(* IEC 61131-3 sources: SRCI/RobotLibrary/Library/POUs/Additional/MC_OpenBrake, 1 file *)

(* ---- MC_OpenBrakeFB.st ---- *)
/// Release robot arm’s brakes.
FUNCTION_BLOCK MC_OpenBrakeFB EXTENDS RobotLibraryBaseExecuteFB
// -------------------------------------------------------------------------
//  SRCI Robot Library
// -------------------------------------------------------------------------
//
//  Object:      OpenBrakeFB
//  Author:      Thorsten Brach
//  Date:        2024-06-01
//
//  Description:
//
//
//  Copyright:
//    (C) 2024 Thorsten Brach. All rights reserved
//             Licensed under the LGPL-3.0 license.
//
//  Disclaimer:
//    This project is provided without any guarantee and can be used for
//    private and commercial purposes. Any use is at the user’s
//    own risk and responsibility.
//
// -------------------------------------------------------------------------
VAR_INPUT
  /// Command parameter
  ParCmd             : OpenBrakeParCmd;
END_VAR

VAR_OUTPUT
  /// Command is transferred and confirmed by the RC
  CommandBuffered   : BOOL;
  /// Receiving of input parameter values has been acknowledged by RC
  ParameterAccepted : BOOL;
  /// Command output
  OutCmd            : OpenBrakeOutCmd;
END_VAR

VAR
  /// internal copy of command parameter
 _parCmd             : OpenBrakeParCmd;
  /// command data to send
 _command            : OpenBrakeSendData;
  /// response data received
 _response           : OpenBrakeRecvData;
END_VAR

  SUPER^(AxesGroup := AxesGroup);

END_FUNCTION_BLOCK

METHOD INTERNAL CheckAddParameter : BOOL
VAR_INPUT
  /// Payload pointer
  PayloadPtr : UDINT;
END_VAR
VAR
  /// Payload as byte array
  Payload    : ARRAY [1..SIZEOF(_command)] OF BYTE;
  /// Null Byte array
  Null       : ARRAY [1..SIZEOF(_command)] OF BYTE;
  /// Data length to compare
  DataLen    : UDINT;
END_VAR

  // Payload pointer must be decreased by one byte, because ADR(Payload) is already one byte !
  PayloadPtr := LIMIT (0, PayloadPtr - 1, SIZEOF(Payload) -1);
  // Convert command struct to payload array
  SysDepMemCpy( pDest := ADR(Payload), pSrc := ADR(_command), DataLen := SIZEOF(_command));
  // Calculate the data length to compare - at least one byte must be compared !
  DataLen := LIMIT(1, SIZEOF(Payload) - PayloadPtr, SIZEOF(Payload));
  // Compare Payload-Array with Null-Byte-Array
  CheckAddParameter := SysDepMemCmp( pData1 := ADR(Payload) + PayloadPtr , pData2 := ADR(Null), DataLen := DataLen) <>  RobotLibraryConstants.OK ;

END_METHOD

METHOD PROTECTED CheckFunctionSupported : BOOL
VAR_IN_OUT
  /// Robot assignment of function
  AxesGroup : AxesGroup;
END_VAR

  CheckFunctionSupported := AxesGroup.State.RobotData.RCSupportedFunctions.OpenBrake;

  IF ( NOT CheckFunctionSupported )
  THEN
    // call base implementation for set error and create log entry
    SUPER^.CheckFunctionSupported(AxesGroup := AxesGroup);
  END_IF

END_METHOD

METHOD PROTECTED CheckParameterChanged : BOOL
VAR_IN_OUT
  /// Robot assignment of function
  AxesGroup    : AxesGroup;
END_VAR

  // Check ParCmd Size is > 0, because MemCmp does not work correctly with size = 0
  IF (SIZEOF(ParCmd) = 0) OR (_stepCmd = 0)
  THEN
    RETURN;
  END_IF

  // compare memory
  _parameterChanged := ( SysDepMemCmp(pData1 := ADR(ParCmd), pData2 := ADR(_parCmd), DataLen := SIZEOF(ParCmd)) <> RobotLibraryConstants.OK );

  // check parameter valid ?
  _parameterValid   := CheckParameterValid( AxesGroup := AxesGroup );

  IF ((  _parameterChanged        )  AND
      (  _parameterValid          )) OR
      (  _parameterUpdateInternal )
  THEN
    // reset internal flag for send parameter update
   _parameterUpdateInternal := FALSE;
    // update internal copy of parameters
   _parCmd := ParCmd;
    // inc parameter sequence
   _command.ParSeq := _command.ParSeq + 1;
    // update command data
    CommandData := CreateCommandPayload(AxesGroup := AxesGroup); // ( Access via reference to rCommandFB in ACR )
    // notify active command register
    AxesGroup.Acyclic.ActiveCommandRegister.NotifyParameterChanged := _uniqueID;
    // Reset parameter accepted flag
    ParameterAccepted := FALSE;
  END_IF

END_METHOD

METHOD PROTECTED CheckParameterValid : BOOL
VAR_IN_OUT
  /// Robot assignment of function
  AxesGroup : AxesGroup;
END_VAR

  CheckParameterValid := TRUE;

  // Check ParCmd.ParCmd.RobotAxesBrakeRelease.AxisJ1 valid ?
  IF (( ParCmd.RobotAxesBrakeRelease.AxisJ1) AND ( NOT AxesGroup.State.RobotData.AxisJointUsed.J1 ))
  THEN
    // Parameter not valid
    CheckParameterValid := FALSE;
    // Set error
    ErrorID := RobotLibraryErrorIdEnum.ERR_INVALID_PAR_CMD;
    // Create log entry
    CreateLogMessagePara1 ( Timestamp   := AxesGroup.State.SystemTime,
                            MessageType := MessageType.CMD,
                            Severity    := Severity.ERROR,
                            MessageCode := ErrorID,
                            MessageText := 'Invalid Parameter ParCmd.RobotAxesBrakeRelease.AxisJ1 = {1}',
                            Para1       :=  BOOL_TO_STRING(ParCmd.RobotAxesBrakeRelease.AxisJ1));
    RETURN;
  END_IF

  // Check ParCmd.ParCmd.RobotAxesBrakeRelease.AxisJ2 valid ?
  IF (( ParCmd.RobotAxesBrakeRelease.AxisJ2) AND ( NOT AxesGroup.State.RobotData.AxisJointUsed.J2 ))
  THEN
    // Parameter not valid
    CheckParameterValid := FALSE;
    // Set error
    ErrorID := RobotLibraryErrorIdEnum.ERR_INVALID_PAR_CMD;
    // Create log entry
    CreateLogMessagePara1 ( Timestamp   := AxesGroup.State.SystemTime,
                            MessageType := MessageType.CMD,
                            Severity    := Severity.ERROR,
                            MessageCode := ErrorID,
                            MessageText := 'Invalid Parameter ParCmd.RobotAxesBrakeRelease.AxisJ2 = {1}',
                            Para1       :=  BOOL_TO_STRING(ParCmd.RobotAxesBrakeRelease.AxisJ2));
    RETURN;
  END_IF

  // Check ParCmd.ParCmd.RobotAxesBrakeRelease.AxisJ3 valid ?
  IF (( ParCmd.RobotAxesBrakeRelease.AxisJ3) AND ( NOT AxesGroup.State.RobotData.AxisJointUsed.J3 ))
  THEN
    // Parameter not valid
    CheckParameterValid := FALSE;
    // Set error
    ErrorID := RobotLibraryErrorIdEnum.ERR_INVALID_PAR_CMD;
    // Create log entry
    CreateLogMessagePara1 ( Timestamp   := AxesGroup.State.SystemTime,
                            MessageType := MessageType.CMD,
                            Severity    := Severity.ERROR,
                            MessageCode := ErrorID,
                            MessageText := 'Invalid Parameter ParCmd.RobotAxesBrakeRelease.AxisJ3 = {1}',
                            Para1       :=  BOOL_TO_STRING(ParCmd.RobotAxesBrakeRelease.AxisJ3));
    RETURN;
  END_IF

  // Check ParCmd.ParCmd.RobotAxesBrakeRelease.AxisJ4 valid ?
  IF (( ParCmd.RobotAxesBrakeRelease.AxisJ4) AND ( NOT AxesGroup.State.RobotData.AxisJointUsed.J4 ))
  THEN
    // Parameter not valid
    CheckParameterValid := FALSE;
    // Set error
    ErrorID := RobotLibraryErrorIdEnum.ERR_INVALID_PAR_CMD;
    // Create log entry
    CreateLogMessagePara1 ( Timestamp   := AxesGroup.State.SystemTime,
                            MessageType := MessageType.CMD,
                            Severity    := Severity.ERROR,
                            MessageCode := ErrorID,
                            MessageText := 'Invalid Parameter ParCmd.RobotAxesBrakeRelease.AxisJ4 = {1}',
                            Para1       :=  BOOL_TO_STRING(ParCmd.RobotAxesBrakeRelease.AxisJ4));
    RETURN;
  END_IF

  // Check ParCmd.ParCmd.RobotAxesBrakeRelease.AxisJ5 valid ?
  IF (( ParCmd.RobotAxesBrakeRelease.AxisJ5) AND ( NOT AxesGroup.State.RobotData.AxisJointUsed.J5 ))
  THEN
    // Parameter not valid
    CheckParameterValid := FALSE;
    // Set error
    ErrorID := RobotLibraryErrorIdEnum.ERR_INVALID_PAR_CMD;
    // Create log entry
    CreateLogMessagePara1 ( Timestamp   := AxesGroup.State.SystemTime,
                            MessageType := MessageType.CMD,
                            Severity    := Severity.ERROR,
                            MessageCode := ErrorID,
                            MessageText := 'Invalid Parameter ParCmd.RobotAxesBrakeRelease.AxisJ5 = {1}',
                            Para1       :=  BOOL_TO_STRING(ParCmd.RobotAxesBrakeRelease.AxisJ5));
    RETURN;
  END_IF

  // Check ParCmd.ParCmd.RobotAxesBrakeRelease.AxisJ6 valid ?
  IF (( ParCmd.RobotAxesBrakeRelease.AxisJ6) AND ( NOT AxesGroup.State.RobotData.AxisJointUsed.J6 ))
  THEN
    // Parameter not valid
    CheckParameterValid := FALSE;
    // Set error
    ErrorID := RobotLibraryErrorIdEnum.ERR_INVALID_PAR_CMD;
    // Create log entry
    CreateLogMessagePara1 ( Timestamp   := AxesGroup.State.SystemTime,
                            MessageType := MessageType.CMD,
                            Severity    := Severity.ERROR,
                            MessageCode := ErrorID,
                            MessageText := 'Invalid Parameter ParCmd.RobotAxesBrakeRelease.AxisJ6 = {1}',
                            Para1       :=  BOOL_TO_STRING(ParCmd.RobotAxesBrakeRelease.AxisJ6));
    RETURN;
  END_IF

  // Check ParCmd.ParCmd.ExternalAxesBrakeRelease.AxisE1 valid ?
  IF (( ParCmd.ExternalAxesBrakeRelease.AxisE1) AND ( NOT AxesGroup.State.RobotData.AxisExternalUsed.E1 ))
  THEN
    // Parameter not valid
    CheckParameterValid := FALSE;
    // Set error
    ErrorID := RobotLibraryErrorIdEnum.ERR_INVALID_PAR_CMD;
    // Create log entry
    CreateLogMessagePara1 ( Timestamp   := AxesGroup.State.SystemTime,
                            MessageType := MessageType.CMD,
                            Severity    := Severity.ERROR,
                            MessageCode := ErrorID,
                            MessageText := 'Invalid Parameter ParCmd.ExternalAxesBrakeRelease.AxisE1 = {1}',
                            Para1       :=  BOOL_TO_STRING(ParCmd.ExternalAxesBrakeRelease.AxisE1));
    RETURN;
  END_IF

  // Check ParCmd.ParCmd.ExternalAxesBrakeRelease.AxisE2 valid ?
  IF (( ParCmd.ExternalAxesBrakeRelease.AxisE2) AND ( NOT AxesGroup.State.RobotData.AxisExternalUsed.E2 ))
  THEN
    // Parameter not valid
    CheckParameterValid := FALSE;
    // Set error
    ErrorID := RobotLibraryErrorIdEnum.ERR_INVALID_PAR_CMD;
    // Create log entry
    CreateLogMessagePara1 ( Timestamp   := AxesGroup.State.SystemTime,
                            MessageType := MessageType.CMD,
                            Severity    := Severity.ERROR,
                            MessageCode := ErrorID,
                            MessageText := 'Invalid Parameter ParCmd.ExternalAxesBrakeRelease.AxisE2 = {1}',
                            Para1       :=  BOOL_TO_STRING(ParCmd.ExternalAxesBrakeRelease.AxisE2));
    RETURN;
  END_IF

  // Check ParCmd.ParCmd.ExternalAxesBrakeRelease.AxisE3 valid ?
  IF (( ParCmd.ExternalAxesBrakeRelease.AxisE3) AND ( NOT AxesGroup.State.RobotData.AxisExternalUsed.E3 ))
  THEN
    // Parameter not valid
    CheckParameterValid := FALSE;
    // Set error
    ErrorID := RobotLibraryErrorIdEnum.ERR_INVALID_PAR_CMD;
    // Create log entry
    CreateLogMessagePara1 ( Timestamp   := AxesGroup.State.SystemTime,
                            MessageType := MessageType.CMD,
                            Severity    := Severity.ERROR,
                            MessageCode := ErrorID,
                            MessageText := 'Invalid Parameter ParCmd.ExternalAxesBrakeRelease.AxisE3 = {1}',
                            Para1       :=  BOOL_TO_STRING(ParCmd.ExternalAxesBrakeRelease.AxisE3));
    RETURN;
  END_IF

  // Check ParCmd.ParCmd.ExternalAxesBrakeRelease.AxisE4 valid ?
  IF (( ParCmd.ExternalAxesBrakeRelease.AxisE4) AND ( NOT AxesGroup.State.RobotData.AxisExternalUsed.E4 ))
  THEN
    // Parameter not valid
    CheckParameterValid := FALSE;
    // Set error
    ErrorID := RobotLibraryErrorIdEnum.ERR_INVALID_PAR_CMD;
    // Create log entry
    CreateLogMessagePara1 ( Timestamp   := AxesGroup.State.SystemTime,
                            MessageType := MessageType.CMD,
                            Severity    := Severity.ERROR,
                            MessageCode := ErrorID,
                            MessageText := 'Invalid Parameter ParCmd.ExternalAxesBrakeRelease.AxisE4 = {1}',
                            Para1       :=  BOOL_TO_STRING(ParCmd.ExternalAxesBrakeRelease.AxisE4));
    RETURN;
  END_IF

  // Check ParCmd.ParCmd.ExternalAxesBrakeRelease.AxisE5 valid ?
  IF (( ParCmd.ExternalAxesBrakeRelease.AxisE5) AND ( NOT AxesGroup.State.RobotData.AxisExternalUsed.E5 ))
  THEN
    // Parameter not valid
    CheckParameterValid := FALSE;
    // Set error
    ErrorID := RobotLibraryErrorIdEnum.ERR_INVALID_PAR_CMD;
    // Create log entry
    CreateLogMessagePara1 ( Timestamp   := AxesGroup.State.SystemTime,
                            MessageType := MessageType.CMD,
                            Severity    := Severity.ERROR,
                            MessageCode := ErrorID,
                            MessageText := 'Invalid Parameter ParCmd.ExternalAxesBrakeRelease.AxisE5 = {1}',
                            Para1       :=  BOOL_TO_STRING(ParCmd.ExternalAxesBrakeRelease.AxisE5));
    RETURN;
  END_IF

  // Check ParCmd.ParCmd.ExternalAxesBrakeRelease.AxisE6 valid ?
  IF (( ParCmd.ExternalAxesBrakeRelease.AxisE6) AND ( NOT AxesGroup.State.RobotData.AxisExternalUsed.E6 ))
  THEN
    // Parameter not valid
    CheckParameterValid := FALSE;
    // Set error
    ErrorID := RobotLibraryErrorIdEnum.ERR_INVALID_PAR_CMD;
    // Create log entry
    CreateLogMessagePara1 ( Timestamp   := AxesGroup.State.SystemTime,
                            MessageType := MessageType.CMD,
                            Severity    := Severity.ERROR,
                            MessageCode := ErrorID,
                            MessageText := 'Invalid Parameter ParCmd.ExternalAxesBrakeRelease.AxisE6 = {1}',
                            Para1       :=  BOOL_TO_STRING(ParCmd.ExternalAxesBrakeRelease.AxisE6));
    RETURN;
  END_IF

END_METHOD

METHOD INTERNAL CreateCommandPayload : RobotLibraryCommandDataFB
VAR_IN_OUT
  /// Robot assignment of function
  AxesGroup : AxesGroup;
END_VAR
VAR
  /// Parameter count
 _parameterCnt : DINT;
END_VAR
// Table 6-681: Sent CMD payload (PLC to RC) of "OpenBrake"
// --------------------------
// Header
// --------------------------
// Byte 00 : UINT  - Type HB
// Byte 01 :       - Type LB
// Byte 02 : USINT - Reserve | ExecutionMode
// Byte 03 : USINT - ParSeq  | Priority
// --------------------------
// Datablock
// --------------------------
// Byte 04 : BYTE  - RobotAxesBrakeRelease
// Byte 05 : BYTE  - ExternalAxesBrakeRelease
// --------------------------

  // set command parameter
  _command.CmdTyp                     :=  CmdType.OpenBrake;
  _command.ExecMode                   :=  ExecMode;
  _command.ParSeq                     := _command.ParSeq;
  _command.Priority                   :=  Priority;
  _command.RobotAxesBrakeRelease.0    := _parCmd.RobotAxesBrakeRelease   .Bit00;
  _command.RobotAxesBrakeRelease.1    := _parCmd.RobotAxesBrakeRelease   .AxisJ1;
  _command.RobotAxesBrakeRelease.2    := _parCmd.RobotAxesBrakeRelease   .AxisJ2;
  _command.RobotAxesBrakeRelease.3    := _parCmd.RobotAxesBrakeRelease   .AxisJ3;
  _command.RobotAxesBrakeRelease.4    := _parCmd.RobotAxesBrakeRelease   .AxisJ4;
  _command.RobotAxesBrakeRelease.5    := _parCmd.RobotAxesBrakeRelease   .AxisJ5;
  _command.RobotAxesBrakeRelease.6    := _parCmd.RobotAxesBrakeRelease   .AxisJ6;
  _command.RobotAxesBrakeRelease.7    := _parCmd.RobotAxesBrakeRelease   .Bit07;
  _command.ExternalAxesBrakeRelease.0 := _parCmd.ExternalAxesBrakeRelease.Bit00;
  _command.ExternalAxesBrakeRelease.1 := _parCmd.ExternalAxesBrakeRelease.AxisE1;
  _command.ExternalAxesBrakeRelease.2 := _parCmd.ExternalAxesBrakeRelease.AxisE2;
  _command.ExternalAxesBrakeRelease.3 := _parCmd.ExternalAxesBrakeRelease.AxisE3;
  _command.ExternalAxesBrakeRelease.4 := _parCmd.ExternalAxesBrakeRelease.AxisE4;
  _command.ExternalAxesBrakeRelease.5 := _parCmd.ExternalAxesBrakeRelease.AxisE5;
  _command.ExternalAxesBrakeRelease.6 := _parCmd.ExternalAxesBrakeRelease.AxisE6;
  _command.ExternalAxesBrakeRelease.7 := _parCmd.ExternalAxesBrakeRelease.Bit07;

  // copy command data to header
  _cmdHeader := _command;
  // call base implementation to copy header to payload buffer
  CreateCommandPayload := SUPER^.CreateCommandPayload(AxesGroup := AxesGroup);

  // Check parameter must be added ?
  IF ( CheckAddParameter(CreateCommandPayload.PayloadPtr))
  THEN
    // add command.RobotAxesBrakeRelease
    CreateCommandPayload.AddByte(_command.RobotAxesBrakeRelease);
    // inc parameter counter
   _parameterCnt := _parameterCnt + 1;
  END_IF

  // Check parameter must be added ?
  IF ( CheckAddParameter(CreateCommandPayload.PayloadPtr))
  THEN
    // add command.ExternalAxesBrakeRelease
    CreateCommandPayload.AddByte(_command.ExternalAxesBrakeRelease);
    // inc parameter counter
   _parameterCnt := _parameterCnt + 1;
  END_IF

  // Create logging
  CreateCommandPayloadLog(AxesGroup := AxesGroup, ParameterCnt := _parameterCnt);

END_METHOD

METHOD INTERNAL CreateCommandPayloadLog
VAR_IN_OUT
  /// Robot assignment of function
  AxesGroup : AxesGroup;
END_VAR
VAR_INPUT
  /// Parameter count
  ParameterCnt : DINT;
END_VAR

  // Create log entry for Parameter start
  CreateLogMessagePara1 ( Timestamp   := AxesGroup.State.SystemTime,
                          MessageType := MessageType.CMD,
                          Severity    := Severity.DEBUG,
                          MessageCode := 0,
                          MessageText := 'Create command payload with the {1} parameter(s) :',
                          Para1       := DINT_TO_STRING(ParameterCnt));

  // Return if no parameter is remaining...
  IF ( ParameterCnt = 0 ) THEN RETURN; END_IF
  // dec remaining parameter(s)
  ParameterCnt := ParameterCnt - 1;
  // Create log entry for RobotAxesBrakeRelease
  CreateLogMessagePara1 ( Timestamp   := AxesGroup.State.SystemTime,
                          MessageType := MessageType.CMD,
                          Severity    := Severity.DEBUG,
                          MessageCode := 0,
                          MessageText := 'Command.RobotAxesBrakeRelease = {1}',
                          Para1       :=  BYTE_TO_STRING_BIN(_command.RobotAxesBrakeRelease));

  // Return if no parameter is remaining...
  IF ( ParameterCnt = 0 ) THEN RETURN; END_IF
  // dec remaining parameter(s)
  ParameterCnt := ParameterCnt - 1;
  // Create log entry for ExternalAxesBrakeRelease
  CreateLogMessagePara1 ( Timestamp   := AxesGroup.State.SystemTime,
                          MessageType := MessageType.CMD,
                          Severity    := Severity.DEBUG,
                          MessageCode := 0,
                          MessageText := 'Command.ExternalAxesBrakeRelease = {1}',
                          Para1       :=  BYTE_TO_STRING_BIN(_command.ExternalAxesBrakeRelease));

END_METHOD

METHOD FB_init : BOOL
VAR_INPUT
  /// if TRUE, the retain variables are initialized (warm start / cold start)
  bInitRetains : BOOL;
  /// if TRUE, the instance afterwards gets moved into the copy code (online change)
  bInCopyCode  : BOOL;
END_VAR

  MyType := 'MC_OpenBrakeFB';

  ExecMode := ExecutionMode.PARALLEL;
  Priority := PriorityLevel.NORMAL;

END_METHOD

METHOD PROTECTED OnExecRun : DINT
VAR_IN_OUT
  /// Robot assignment of function
  AxesGroup : AxesGroup;
END_VAR

  // call base implementation
  SUPER^.OnExecRun(AxesGroup := AxesGroup);

  CASE _stepCmd OF

    00:  IF ( _execute_R.Q ) AND ( NOT Error)
         THEN
           // Check function is supported and parameter are valid ?
           IF (( CheckFunctionSupported( AxesGroup := AxesGroup )) AND
               ( CheckParameterValid   ( AxesGroup := AxesGroup )))
           THEN
             // set busy flag
             Busy := TRUE;
             // Reset command outputs
             SysDepMemSet(pDest := ADR(OutCmd), Value := 0, DataLen := SIZEOF(OutCmd));
             // apply command parameter
            _parCmd := ParCmd;
             // init parameter sequence
            _command.ParSeq := 1;
             // create command data
             CommandData := CreateCommandPayload(AxesGroup := AxesGroup);
             // Add command to active command register
            _uniqueID := AxesGroup.Acyclic.ActiveCommandRegister.AddCmd( pCommandFB := ADR(THIS^ ));
             // set timeout
             SetTimeout(PT := _timeoutCmd, rTimer := _timerCmd);
             // inc step counter
            _stepCmd := _stepCmd + 1;
           END_IF
         END_IF

    01:  // Wait for responce received
         IF ( _responseReceived )
         THEN
           // reset response received flag
          _responseReceived := FALSE;

           CASE  _response.State
           OF
             CmdMessageState.BUFFERED    : CommandBuffered    := TRUE;
             CmdMessageState.ACTIVE      : ParameterAccepted  := TRUE;
             CmdMessageState.DONE        : Done               := TRUE;
             CmdMessageState.ERROR       : Error              := TRUE;
           END_CASE

           // Done, Aborted or Error ?
           IF (_response.State >= CmdMessageState.DONE )
           THEN
             // Reset Busy flag
             Busy := FALSE;
             // Update results
             OutCmd.Enabled                          := _response.Enabled.0;
             OutCmd.RobotAxesBrakeReleased.Bit00     := _response.RobotAxesBrakeReleased.0;
             OutCmd.RobotAxesBrakeReleased.AxisJ1    := _response.RobotAxesBrakeReleased.1;
             OutCmd.RobotAxesBrakeReleased.AxisJ2    := _response.RobotAxesBrakeReleased.2;
             OutCmd.RobotAxesBrakeReleased.AxisJ3    := _response.RobotAxesBrakeReleased.3;
             OutCmd.RobotAxesBrakeReleased.AxisJ4    := _response.RobotAxesBrakeReleased.4;
             OutCmd.RobotAxesBrakeReleased.AxisJ5    := _response.RobotAxesBrakeReleased.5;
             OutCmd.RobotAxesBrakeReleased.AxisJ6    := _response.RobotAxesBrakeReleased.6;
             OutCmd.RobotAxesBrakeReleased.Bit07     := _response.RobotAxesBrakeReleased.7;
             OutCmd.ExternalAxesBrakeReleased.Bit00  := _response.ExternalAxesBrakeReleased.0;
             OutCmd.ExternalAxesBrakeReleased.AxisE1 := _response.ExternalAxesBrakeReleased.1;
             OutCmd.ExternalAxesBrakeReleased.AxisE2 := _response.ExternalAxesBrakeReleased.2;
             OutCmd.ExternalAxesBrakeReleased.AxisE3 := _response.ExternalAxesBrakeReleased.3;
             OutCmd.ExternalAxesBrakeReleased.AxisE4 := _response.ExternalAxesBrakeReleased.4;
             OutCmd.ExternalAxesBrakeReleased.AxisE5 := _response.ExternalAxesBrakeReleased.5;
             OutCmd.ExternalAxesBrakeReleased.AxisE6 := _response.ExternalAxesBrakeReleased.6;
             OutCmd.ExternalAxesBrakeReleased.Bit07  := _response.ExternalAxesBrakeReleased.7;

             // set timeout
             SetTimeout(PT := _timeoutCmd, rTimer := _timerCmd);
             // inc step counter
            _stepCmd := _stepCmd + 1;
           END_IF
         END_IF

    02: IF ( NOT Execute)
        THEN
          Reset();
        END_IF
  ELSE
    // invalid step
    ErrorID := RobotLibraryErrorIdEnum.ERR_INVALID_STEP;
  END_CASE

  // Reset FB
  IF ( NOT Execute )
  THEN
    Reset();
  END_IF

END_METHOD

METHOD INTERNAL ParseResponsePayload : DINT
VAR_INPUT
  /// Response data
  ResponseData : RobotLibraryResponseDataFB;
  /// Timestamp
  Timestamp    : SystemTime;
END_VAR
VAR
  /// Parameter count
 _parameterCnt : DINT;
END_VAR
// Table 6-682: Received CMD payload (RC to PLC) of "OpenBrake"
// --------------------------
// Header
// --------------------------
// Byte 00 : USINT - ParSeq | State
// Byte 01 : SINT  - AlarmMessageSeverity
// Byte 02 : UINT  - AlarmMessageCode HB
// Byte 03 :       - AlarmMessageCode LB
// --------------------------
// Datablock
// --------------------------
// Byte 04 : BOOL  - Enabled
// Byte 05 : BYTE  - RobotAxesBrakeReleased
// Byte 06 : BYTE  - ExternalAxesBrakeReleased
// --------------------------

  // call base implementation to parse the header from payload buffer
  ResponseData.PayloadPtr := SUPER^.ParseResponsePayload(ResponseData := ResponseData, Timestamp := Timestamp);

  // copy parsed header to response
  _response.ParSeq               := _rspHeader.ParSeq;
  _response.State                := _rspHeader.State;
  _response.AlarmMessageSeverity := _rspHeader.AlarmMessageSeverity;
  _response.AlarmMessageCode     := _rspHeader.AlarmMessageCode;

  // Check payload remaining ?
  IF ( ResponseData.IsPayloadRemaining)
  THEN
    // Get RobotAxesStatus
   _response.RobotAxesBrakeReleased := ResponseData.GetByte();
    // inc parameter counter
   _parameterCnt := _parameterCnt + 1;
  END_IF

  // Check payload remaining ?
  IF ( ResponseData.IsPayloadRemaining)
  THEN
    // Get ExternalAxesStatus
   _response.ExternalAxesBrakeReleased := ResponseData.GetByte();
    // inc parameter counter
   _parameterCnt := _parameterCnt + 1;
  END_IF

  // Create logging
  ParseResponsePayloadLog(ResponseData := ResponseData, Timestamp := Timestamp, ParameterCnt := _parameterCnt);

END_METHOD

METHOD INTERNAL ParseResponsePayloadLog
VAR_INPUT
  /// Response data
  ResponseData : RobotLibraryResponseDataFB;
  /// Timestamp
  Timestamp    : SystemTime;
  /// Parameter count
  ParameterCnt : DINT;
END_VAR

  // Create log entry for Parameter start
  CreateLogMessagePara1 ( Timestamp   := Timestamp,
                          MessageType := MessageType.CMD,
                          Severity    := Severity.DEBUG,
                          MessageCode := 0,
                          MessageText := '{1} parameter(s) to parse from the response data:',
                          Para1       := DINT_TO_STRING(ParameterCnt));

  // Return if no parameter is remaining...
  IF ( ParameterCnt = 0 ) THEN RETURN; END_IF
  // dec remaining parameter(s)
  ParameterCnt := ParameterCnt - 1;
  // Create log entry for RobotAxesBrakeReleased
  CreateLogMessagePara1 ( Timestamp   := Timestamp,
                          MessageType := MessageType.CMD,
                          Severity    := Severity.DEBUG,
                          MessageCode := 0,
                          MessageText := 'Response.RobotAxesBrakeReleased = {1}',
                          Para1       :=  BYTE_TO_STRING_BIN(_response.RobotAxesBrakeReleased));

  // Return if no parameter is remaining...
  IF ( ParameterCnt = 0 ) THEN RETURN; END_IF
  // dec remaining parameter(s)
  ParameterCnt := ParameterCnt - 1;
  // Create log entry for ExternalAxesBrakeReleased
  CreateLogMessagePara1 ( Timestamp   := Timestamp,
                          MessageType := MessageType.CMD,
                          Severity    := Severity.DEBUG,
                          MessageCode := 0,
                          MessageText := 'Response.ExternalAxesBrakeReleased = {1}',
                          Para1       :=  BYTE_TO_STRING_BIN(_response.ExternalAxesBrakeReleased));

END_METHOD

METHOD PROTECTED Reset : DINT
VAR_INPUT
END_VAR

  Reset := SUPER^.Reset();

  Done               := FALSE;
  Busy               := FALSE;
  CommandBuffered    := FALSE;
  ParameterAccepted  := FALSE;

END_METHOD
